% RSLogix 500 project PRACTISE-17.RSS, saved by version 8.30.00.16 %
PROJECT "UNTITLED"    % processor: MicroLogix 1000 %

PROGRAM FILES
  LAD 2 "MAIN_PROG"  8 rungs
  LAD 3 "USER_FAULT"  1 rungs
  LAD 4 "HSC_INT"  1 rungs
  LAD 5 "STI_INT"  1 rungs
  LAD 6, 7, 8, 9, 10, 11, 12, 13, 14, 15, 16: only END

DATA FILES
  O0 OUTPUT  1 elements
  I1 INPUT  2 elements
  S2 STATUS  33 elements
  B3 BINARY  32 elements
  T4 TIMER  40 elements
  C5 COUNTER  32 elements
  R6 CONTROL  16 elements
  N7 INTEGER  105 elements

LADDER 2 "MAIN_PROG"
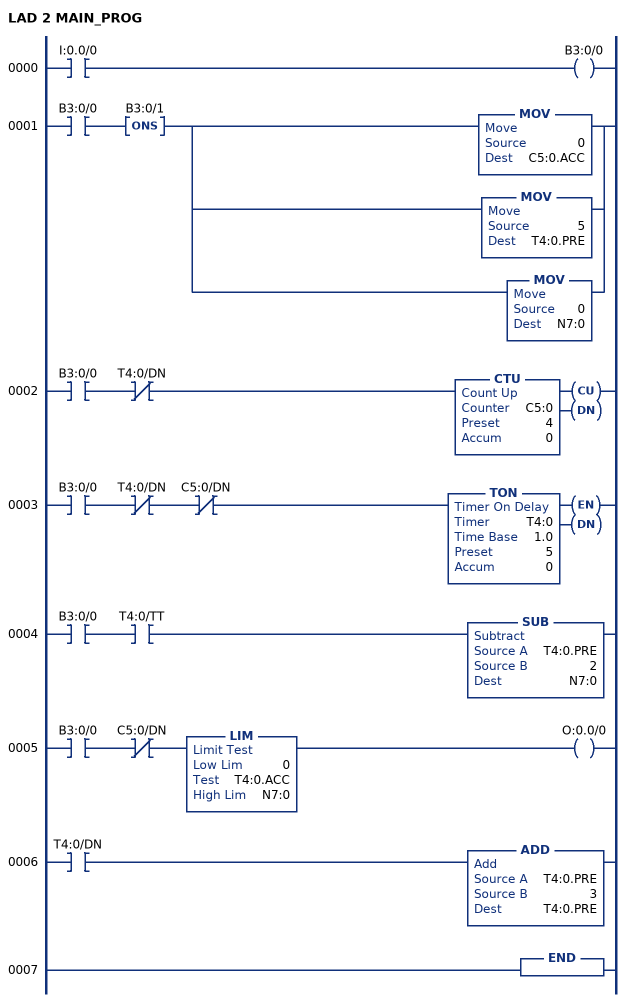
% Rung: 0 %
SOR XIC I:0.0/0 OTE B3:0/0 EOR
% Rung: 1 %
SOR XIC B3:0/0 OSR B3:0/1 BST MOV 0 C5:0.ACC NXB BST MOV 5 T4:0.PRE NXB MOV 0 N7:0 BND BND EOR
% Rung: 2 %
SOR XIC B3:0/0 XIO T4:0/DN CTU C5:0 4 0 EOR
% Rung: 3 %
SOR XIC B3:0/0 XIO T4:0/DN XIO C5:0/DN TON T4:0 1.0 5 0 EOR
% Rung: 4 %
SOR XIC B3:0/0 XIC T4:0/TT SUB T4:0.PRE 2 N7:0 EOR
% Rung: 5 %
SOR XIC B3:0/0 XIO C5:0/DN LIM 0 T4:0.ACC N7:0 OTE O:0.0/0 EOR
% Rung: 6 %
SOR XIC T4:0/DN ADD T4:0.PRE 3 T4:0.PRE EOR
% Rung: 7 %
SOR END EOR

DATA TABLE (non-zero values as saved)
DATA T4
% .PRE .ACC %
% T4:0 % 5 0
DATA C5
% .PRE .ACC %
% C5:0 % 4 0
DATA N7
% N7:0 % 12 0 0 0 0 0 0 0 0 0
